Universal Robots PolyScope program: ros.urp

Program ros (installation=default directory=/ursim/programs createdIn=5.4.2.76197 lastSavedIn=5.4.2.76197 robotSerialNumber=20183099999)
Calibrated DH parameters: a=[0, -0.6127, -0.57155, 0, 0, 0]; d=[0.1807, 0, 0, 0.17415, 0.11985, 0.11655]; alpha=[1.570796, 0, 0, 1.570796, -1.570796, 0]; deltaTheta=[0, 0, 0, 0, 0, 0]
Robot Program (runOnlyOnce=false)
  URCap External Control (External Control, FZI Research Center for Information Technology)
